Staubli VAL3: send_data.pgx

program send_data()
  local string snd_msg
  local num i
  local num nSent
begin

  putln("Start to send data !")

  do

  snd_msg = toString(".4",getSpeed(tTool)) + chr(13) + chr(10)

  for i=0 to len(snd_msg)-1
    nSent = sioSet(sioASCII,asc(snd_msg,i))

    if nSent != 1
      check_status = false
      stopMove()
      cls()
      putln("Communication error !")
      disablePower()
    endIf


  endFor

  //putln(snd_msg)

  //cls()
  delay(.2)

  until check_status != true


end
